// TIA Portal V18 export
DATA_BLOCK "Control"   // DB68
{ S7_Optimized_Access := 'TRUE' }
VERSION : 0.1
// stored: AutoNumber true, DBAccessibleFromOPCUA true, IsOnlyStoredInLoadMemory false, IsRetainMemResEnabled false, IsWriteProtectedInAS false, MemoryReserve 100
   VAR
      "waiting For pre run" : Bool := TRUE;
      "ready for operation" : Bool := FALSE;
      "metering blocked" : Bool := FALSE;
      "change Screen" : Int := 0;
      "A metering ready" : Bool := TRUE;
      "B metering ready" : Bool := TRUE;
      "A&B metering ready" : Bool := TRUE;
      "metering program ready" : Bool := FALSE;
      "Evacuation Ready Tank A1" : Bool := FALSE;
      "Evacuation Ready Tank A2" : Bool := FALSE;
      "Evacuation Read" : Bool := FALSE;
      "Recirculation Enabled" : Bool := FALSE;
      "recirculation okay" : Bool := FALSE;
      "Show start Button" : Bool := FALSE;
      "Show esc Button" : Bool := FALSE;
      "Show stop Button" : Bool := FALSE;
      "Do not show para& config button" : Bool := FALSE;
   END_VAR
   VAR RETAIN
      "Start signal on site type" : Int := 1;
      "stop signal on site type" : Int := 0;
      "Program selection Mode" : Int := 0;
      "Flowrate adjustment type" : Int := 0;
   END_VAR
   VAR
      "A recirculation Ready" : Bool := FALSE;
      "B recirculation Ready" : Bool := FALSE;
      "recirculation ready" : Bool := FALSE;
      "Show alarm field" : Bool := FALSE;
      "Flush ready" : Bool := TRUE;
      "ratio check Ready" : Bool := TRUE;
      "reset from hmi _site_pb_PN" : Bool := FALSE;
      "start from hmi_site_pb_PN" : Bool := FALSE;
      "stop from hmi_site_pb_PN" : Bool := FALSE;
      "Heater OK" : Bool := FALSE;
      "Heater No Fault" : Bool := FALSE;
   END_VAR
   VAR RETAIN
      "Pump A maximum Idle Time" : Int := 30;
      "Pump B maximum Idle Time" : Int := 30;
   END_VAR
   VAR
      "Pump A maximum Idle Time sec" : DInt := 1800000;
      "Pump B maximum Idle Time sec" : DInt := 1800000;
      Mute : Struct
         "Mute enable" : Bool := FALSE;
         "Mute buzzer" : Bool := FALSE;
         "Mutte On" : Bool := FALSE;
      END_STRUCT;
      Pressure_sensor_select : Int := 0;
   END_VAR
   VAR RETAIN
      Level_sensor_enable : Bool := FALSE;
      "Minimum Dispesing qty" : Real;
      "Minimum Snuff back qty" : Real;
      "Outlet On_off" : Bool;
   END_VAR
   VAR
      "Outlet On_off_disp" : Bool;
   END_VAR
BEGIN
END_DATA_BLOCK
